(* IEC 61131-3 sources: eCockpitGit/test_project/src/%F%00 Library/%F%JSON/%POU%FB_JSONReader/%F%Internal, 2 files *)

(* ---- %METH%checkNoBackSlash.st ---- *)
//This method checks if there is a backslash in front of the code, then checks if there is an backslash in front of that and so on, if the amount of backslashes is even or if there are none it returns true
// |**Version**|**Author**| **Date** |**Changes**
// | 1         | NSN      | 06-07-20 | Creation
METHOD PROTECTED checkNoBackSlash : BOOL
VAR_INPUT
	checkPos		:POINTER TO EASCII;
END_VAR
VAR
	checkCount		:DWORD;
END_VAR
(*%!%__DELIMITER__%!%*)
IF checkPos > bufferADROrg THEN
	checkPos				:=		checkPos - 1;
	WHILE checkPos^ = EASCII.BackSlash AND_THEN checkPos > bufferADROrg DO
		checkCount			:=		checkCount + 1;
		checkPos			:=		checkPos - 1;
	END_WHILE
	checkNoBackSlash		:=		checkCount MOD 2 = 0;
ELSE
	checkNoBackSlash		:=		TRUE;
END_IF

(* ---- %METH%getType.st ---- *)
//This method checks what type the json value is, it must be given the first byte after the colon
// |**Version**|**Author**| **Date** |**Changes**
// | 1         | NSN      | 04-07-20 | Creation
METHOD PROTECTED getType :EStructType
VAR_INPUT
	valueFirstByte		:POINTER TO EASCII;		//The position to search the json type from
END_VAR
VAR_OUTPUT
	valuePos			:POINTER TO EASCII;		//The actual start of the value after any whitespace
END_VAR
(*%!%__DELIMITER__%!%*)
//Initial result is set as invalid, when json type cannot be determined
getType								:=		EStructType.invalid;
WHILE valueFirstByte <= bufferADRMax DO
	CASE valueFirstByte^ OF
		EASCII.Smallf,EASCII.Smallt:
			valuePos				:=		valueFirstByte;
			getType					:=		EStructType.tBool;
			EXIT;
		EASCII.DoubleQoute:
			valuePos				:=		valueFirstByte;
			getType					:=		EStructType.tString;
			EXIT;
		EASCII.SqBracketO:
			valuePos				:=		valueFirstByte;
			getType					:=		EStructType.tArray;
			EXIT;
		EASCII.OpenBraces:
			valuePos				:=		valueFirstByte;
			getType					:=		EStructType.object;
			EXIT;
		EASCII.Smalln:
			valuePos				:=		valueFirstByte;
			getType					:=		EStructType.null;
			EXIT;
		EASCII.Zero,EASCII.One,EASCII.Two,EASCII.Three,EASCII.Four,EASCII.Five,EASCII.Six,EASCII.Seven,EASCII.Eight,EASCII.Nine,EASCII.Minus:
			valuePos				:=		valueFirstByte;
			getType					:=		EStructType.number;
			EXIT;
		EASCII.SqBracketC,EASCII.CloseBraces:
			getType					:=		EStructType.none;
			EXIT;
	END_CASE
	valueFirstByte					:=		valueFirstByte + 1;
END_WHILE
